LIN {X 0,Y 125.96,Z 856.864,A -85,B 0,C 180,E1 -29175.835,E2 -29175.835} C_VEL
LIN {X 0,Y 122.097,Z 869.522,A -85,B 0,C 180,E1 -29176.604,E2 -29176.604} C_VEL
LIN {X 0,Y 116.788,Z 882.194,A -85,B 0,C 180,E1 -29177.633,E2 -29177.633} C_VEL
LIN {X 0,Y 110.546,Z 893.75,A -85,B 0,C 180,E1 -29179.056,E2 -29179.056} C_VEL
LIN {X 0,Y 103.315,Z 904.432,A -85,B 0,C 180,E1 -29180.801,E2 -29180.801} C_VEL
LIN {X 0,Y 95.494,Z 914.111,A -85,B 0,C 180,E1 -29183.161,E2 -29183.161} C_VEL
LIN {X 0,Y 86.375,Z 923.456,A -85,B 0,C 180,E1 -29186.565,E2 -29186.565} C_VEL
LIN {X 0,Y 77.748,Z 931.029,A -85,B 0,C 180,E1 -29190.898,E2 -29190.898} C_VEL
LIN {X 0,Y 69.801,Z 937.172,A -85,B 0,C 180,E1 -29196.413,E2 -29196.413} C_VEL
LIN {X 0,Y 62.757,Z 942.089,A -85,B 0,C 180,E1 -29203.354,E2 -29203.354} C_VEL
LIN {X 0,Y 56.919,Z 945.911,A -85,B 0,C 180,E1 -29211.938,E2 -29211.938} C_VEL
LIN {X 0,Y 53.931,Z 947.927,A -85,B 0,C 180,E1 -29218.644,E2 -29218.644} C_VEL
LIN {X 0,Y 50.672,Z 950.661,A -85,B 0,C 180,E1 -29233.952,E2 -29233.952} C_VEL
LIN {X 0,Y 50.511,Z 951.445,A -85,B 0,C 180,E1 -29242.056,E2 -29242.056} C_VEL
LIN {X 0,Y 51.125,Z 951.803,A -85,B 0,C 180,E1 -29250.052,E2 -29250.052} C_VEL
LIN {X 0,Y 50.744,Z 950.876,A -85,B 0,C 180,E1 -29264.189,E2 -29264.189} C_VEL
LIN {X 0,Y 52.243,Z 949.486,A -85,B 0,C 180,E1 -29273.856,E2 -29273.856} C_VEL
LIN {X 0,Y 56.006,Z 946.967,A -85,B 0,C 180,E1 -29284.436,E2 -29284.436} C_VEL
LIN {X 0,Y 61.604,Z 943.508,A -85,B 0,C 180,E1 -29293.252,E2 -29293.252} C_VEL
LIN {X 0,Y 68.709,Z 939.048,A -85,B 0,C 180,E1 -29300.154,E2 -29300.154} C_VEL
LIN {X 0,Y 71.326,Z 937.319,A -85,B 0,C 180,E1 -29302.08,E2 -29302.08} C_VEL
LIN {X 0,Y 72.417,Z 935.739,A -85,B 0,C 180,E1 -29304.388,E2 -29304.388} C_VEL
LIN {X 0,Y 64.144,Z 929.643,A -85,B 0,C 180,E1 -29327.342,E2 -29327.342} C_VEL
LIN {X 0,Y 66.621,Z 924.428,A -85,B 0,C 180,E1 -29346.056,E2 -29346.056} C_VEL
LIN {X 0,Y 72.228,Z 920.62,A -85,B 0,C 180,E1 -29356.973,E2 -29356.973} C_VEL
LIN {X 0,Y 79.37,Z 916.695,A -85,B 0,C 180,E1 -29364.251,E2 -29364.251} C_VEL
LIN {X 0,Y 85.958,Z 913.489,A -85,B 0,C 180,E1 -29369.378,E2 -29369.378} C_VEL
LIN {X 0,Y 89.672,Z 911.586,A -85,B 0,C 180,E1 -29371.415,E2 -29371.415} C_VEL
LIN {X 0,Y 88.137,Z 913.443,A -85,B 0,C 180,E1 -29373.098,E2 -29373.098} C_VEL
LIN {X 0,Y 80.195,Z 920.191,A -85,B 0,C 180,E1 -29377.884,E2 -29377.884} C_VEL
LIN {X 0,Y 73.038,Z 925.543,A -85,B 0,C 180,E1 -29383.758,E2 -29383.758} C_VEL
LIN {X 0,Y 68.621,Z 928.473,A -85,B 0,C 180,E1 -29388.214,E2 -29388.214} C_VEL
LIN {X 0,Y 63.119,Z 931.664,A -85,B 0,C 180,E1 -29394.789,E2 -29394.789} C_VEL
LIN {X 0,Y 59.712,Z 933.322,A -85,B 0,C 180,E1 -29399.034,E2 -29399.034} C_VEL
LIN {X 0,Y 53.34,Z 935.711,A -85,B 0,C 180,E1 -29406.365,E2 -29406.365} C_VEL
LIN {X 0,Y 48.796,Z 937.088,A -85,B 0,C 180,E1 -29413.525,E2 -29413.525} C_VEL
LIN {X 0,Y 46.59,Z 937.681,A -85,B 0,C 180,E1 -29420.091,E2 -29420.091} C_VEL
LIN {X 0,Y 46.223,Z 937.775,A -85,B 0,C 180,E1 -29422.482,E2 -29422.482} C_VEL
LIN {X 0,Y 46.353,Z 937.773,A -85,B 0,C 180,E1 -29438.662,E2 -29438.662} C_VEL
LIN {X 0,Y 47.82,Z 937.194,A -85,B 0,C 180,E1 -29447.034,E2 -29447.034} C_VEL
LIN {X 0,Y 52.969,Z 934.956,A -85,B 0,C 180,E1 -29461.993,E2 -29461.993} C_VEL
LIN {X 0,Y 58.863,Z 932.124,A -85,B 0,C 180,E1 -29470.983,E2 -29470.983} C_VEL
LIN {X 0,Y 65.813,Z 928.288,A -85,B 0,C 180,E1 -29478.31,E2 -29478.31} C_VEL
LIN {X 0,Y 74.181,Z 922.798,A -85,B 0,C 180,E1 -29485.018,E2 -29485.018} C_VEL
LIN {X 0,Y 82.984,Z 915.971,A -85,B 0,C 180,E1 -29490.164,E2 -29490.164} C_VEL
LIN {X 0,Y 91.726,Z 907.926,A -85,B 0,C 180,E1 -29494.12,E2 -29494.12} C_VEL
LIN {X 0,Y 99.199,Z 899.686,A -85,B 0,C 180,E1 -29496.996,E2 -29496.996} C_VEL
LIN {X 0,Y 106.833,Z 889.483,A -85,B 0,C 180,E1 -29499.543,E2 -29499.543} C_VEL
LIN {X 0,Y 112.682,Z 880.047,A -85,B 0,C 180,E1 -29501.229,E2 -29501.229} C_VEL
LIN {X 0,Y 117.281,Z 871.144,A -85,B 0,C 180,E1 -29502.419,E2 -29502.419} C_VEL
LIN {X 0,Y 122.094,Z 859.374,A -85,B 0,C 180,E1 -29503.611,E2 -29503.611} C_VEL
LIN {X 0,Y 125.844,Z 846.575,A -85,B 0,C 180,E1 -29504.721,E2 -29504.721} C_VEL
LIN {X 0,Y 127.634,Z 837.303,A -85,B 0,C 180,E1 -29505.399,E2 -29505.399} C_VEL
LIN {X 0,Y 126.554,Z 833.188,A -85,B 0,C 180,E1 -29509.4,E2 -29509.4} C_VEL
LIN {X 0,Y 125.802,Z 830.534,A -85,B 0,C 180,E1 -29513.182,E2 -29513.182} C_VEL
LIN {X 0,Y 125.399,Z 828.562,A -85,B 0,C 180,E1 -29518.394,E2 -29518.394} C_VEL
LIN {X 0,Y 125.412,Z 829.133,A -85,B 0,C 180,E1 -29521.204,E2 -29521.204} C_VEL
LIN {X 0,Y 125.607,Z 830.225,A -85,B 0,C 180,E1 -29523.709,E2 -29523.709} C_VEL
LIN {X 0,Y 126.013,Z 834.743,A -85,B 0,C 180,E1 -29527.511,E2 -29527.511} C_VEL
LIN {X 0,Y 126.597,Z 840.675,A -85,B 0,C 180,E1 -29531.003,E2 -29531.003} C_VEL
LIN {X 0,Y 126.639,Z 841.245,A -85,B 0,C 180,E1 -29531.267,E2 -29531.267} C_VEL
LIN {X 0,Y 124.687,Z 853.794,A -85,B 0,C 180,E1 -29532.524,E2 -29532.524} C_VEL
LIN {X 0,Y 121.012,Z 866.448,A -85,B 0,C 180,E1 -29533.224,E2 -29533.224} C_VEL
LIN {X 0,Y 115.867,Z 878.975,A -85,B 0,C 180,E1 -29534.064,E2 -29534.064} C_VEL
LIN {X 0,Y 109.95,Z 890.23,A -85,B 0,C 180,E1 -29535.191,E2 -29535.191} C_VEL
LIN {X 0,Y 102.648,Z 901.262,A -85,B 0,C 180,E1 -29536.661,E2 -29536.661} C_VEL
LIN {X 0,Y 94.543,Z 911.298,A -85,B 0,C 180,E1 -29538.697,E2 -29538.697} C_VEL
LIN {X 0,Y 85.004,Z 921.052,A -85,B 0,C 180,E1 -29541.64,E2 -29541.64} C_VEL
LIN {X 0,Y 75.838,Z 928.871,A -85,B 0,C 180,E1 -29545.463,E2 -29545.463} C_VEL
LIN {X 0,Y 68.563,Z 934.267,A -85,B 0,C 180,E1 -29549.478,E2 -29549.478} C_VEL
LIN {X 0,Y 60.542,Z 939.563,A -85,B 0,C 180,E1 -29555.731,E2 -29555.731} C_VEL
LIN {X 0,Y 53.518,Z 943.742,A -85,B 0,C 180,E1 -29563.835,E2 -29563.835} C_VEL
LIN {X 0,Y 47.968,Z 946.908,A -85,B 0,C 180,E1 -29574.194,E2 -29574.194} C_VEL
LIN {X 0,Y 43.825,Z 949.638,A -85,B 0,C 180,E1 -29591.358,E2 -29591.358} C_VEL
LIN {X 0,Y 43.425,Z 950.423,A -85,B 0,C 180,E1 -29600.749,E2 -29600.749} C_VEL
LIN {X 0,Y 44.019,Z 950.789,A -85,B 0,C 180,E1 -29610.061,E2 -29610.061} C_VEL
LIN {X 0,Y 43.801,Z 949.941,A -85,B 0,C 180,E1 -29625.697,E2 -29625.697} C_VEL
LIN {X 0,Y 45.805,Z 948.467,A -85,B 0,C 180,E1 -29637.47,E2 -29637.47} C_VEL
LIN {X 0,Y 50.302,Z 945.951,A -85,B 0,C 180,E1 -29649.021,E2 -29649.021} C_VEL
LIN {X 0,Y 56.65,Z 942.495,A -85,B 0,C 180,E1 -29658.171,E2 -29658.171} C_VEL
LIN {X 0,Y 64.087,Z 938.238,A -85,B 0,C 180,E1 -29664.741,E2 -29664.741} C_VEL
LIN {X 0,Y 63.801,Z 937.55,A -85,B 0,C 180,E1 -29666.58,E2 -29666.58} C_VEL
LIN {X 0,Y 57.709,Z 931.539,A -85,B 0,C 180,E1 -29693.005,E2 -29693.005} C_VEL
LIN {X 0,Y 66.173,Z 924.542,A -85,B 0,C 180,E1 -29718.58,E2 -29718.58} C_VEL
LIN {X 0,Y 77.85,Z 919.066,A -85,B 0,C 180,E1 -29729.77,E2 -29729.77} C_VEL
LIN {X 0,Y 79.132,Z 918.523,A -85,B 0,C 180,E1 -29730.709,E2 -29730.709} C_VEL
LIN {X 0,Y 77.189,Z 920.414,A -85,B 0,C 180,E1 -29733.114,E2 -29733.114} C_VEL
LIN {X 0,Y 68.366,Z 926.547,A -85,B 0,C 180,E1 -29739.5,E2 -29739.5} C_VEL
LIN {X 0,Y 63.553,Z 929.477,A -85,B 0,C 180,E1 -29743.988,E2 -29743.988} C_VEL
LIN {X 0,Y 56.806,Z 933.027,A -85,B 0,C 180,E1 -29751.729,E2 -29751.729} C_VEL
LIN {X 0,Y 53.033,Z 934.846,A -85,B 0,C 180,E1 -29757.932,E2 -29757.932} C_VEL
LIN {X 0,Y 47.849,Z 937.141,A -85,B 0,C 180,E1 -29772.86,E2 -29772.86} C_VEL
LIN {X 0,Y 46.223,Z 937.775,A -85,B 0,C 180,E1 -29782.482,E2 -29782.482} C_VEL
LIN {X 0,Y 45.161,Z 938.065,A -85,B 0,C 180,E1 -29789.784,E2 -29789.784} C_VEL
LIN {X 0,Y 43.227,Z 938.129,A -85,B 0,C 180,E1 -29802.443,E2 -29802.443} C_VEL
LIN {X 0,Y 43.031,Z 937.744,A -85,B 0,C 180,E1 -29813.036,E2 -29813.036} C_VEL
LIN {X 0,Y 44.873,Z 936.848,A -85,B 0,C 180,E1 -29821.669,E2 -29821.669} C_VEL
LIN {X 0,Y 45.325,Z 936.617,A -85,B 0,C 180,E1 -29822.768,E2 -29822.768} C_VEL
LIN {X 0,Y 51.399,Z 934.17,A -85,B 0,C 180,E1 -29833.056,E2 -29833.056} C_VEL
LIN {X 0,Y 58.815,Z 930.661,A -85,B 0,C 180,E1 -29840.883,E2 -29840.883} C_VEL
LIN {X 0,Y 68.575,Z 924.982,A -85,B 0,C 180,E1 -29848.511,E2 -29848.511} C_VEL
LIN {X 0,Y 76.72,Z 919.301,A -85,B 0,C 180,E1 -29853.185,E2 -29853.185} C_VEL
LIN {X 0,Y 85.798,Z 911.83,A -85,B 0,C 180,E1 -29857.061,E2 -29857.061} C_VEL
LIN {X 0,Y 93.556,Z 904.17,A -85,B 0,C 180,E1 -29859.793,E2 -29859.793} C_VEL
LIN {X 0,Y 101.396,Z 894.827,A -85,B 0,C 180,E1 -29862.274,E2 -29862.274} C_VEL
LIN {X 0,Y 108.587,Z 884.423,A -85,B 0,C 180,E1 -29864.206,E2 -29864.206} C_VEL
LIN {X 0,Y 114.83,Z 873.288,A -85,B 0,C 180,E1 -29865.58,E2 -29865.58} C_VEL
LIN {X 0,Y 118.787,Z 864.334,A -85,B 0,C 180,E1 -29866.514,E2 -29866.514} C_VEL
LIN {X 0,Y 122.781,Z 852.78,A -85,B 0,C 180,E1 -29867.478,E2 -29867.478} C_VEL
LIN {X 0,Y 125.431,Z 841.744,A -85,B 0,C 180,E1 -29868.317,E2 -29868.317} C_VEL
LIN {X 0,Y 124.898,Z 838.871,A -85,B 0,C 180,E1 -29871.709,E2 -29871.709} C_VEL
LIN {X 0,Y 124.692,Z 837.34,A -85,B 0,C 180,E1 -29873.933,E2 -29873.933} C_VEL
LIN {X 0,Y 124.479,Z 835.709,A -85,B 0,C 180,E1 -29878.382,E2 -29878.382} C_VEL
LIN {X 0,Y 124.49,Z 836.12,A -85,B 0,C 180,E1 -29880.809,E2 -29880.809} C_VEL
LIN {X 0,Y 124.572,Z 837.021,A -85,B 0,C 180,E1 -29882.728,E2 -29882.728} C_VEL
LIN {X 0,Y 124.685,Z 840.698,A -85,B 0,C 180,E1 -29885.864,E2 -29885.864} C_VEL
LIN {X 0,Y 124.757,Z 844.677,A -85,B 0,C 180,E1 -29888.301,E2 -29888.301} C_VEL
LIN {X 0,Y 122.942,Z 854.393,A -85,B 0,C 180,E1 -29889.356,E2 -29889.356} C_VEL
LIN {X 0,Y 119.094,Z 866.746,A -85,B 0,C 180,E1 -29889.963,E2 -29889.963} C_VEL
LIN {X 0,Y 113.682,Z 879.359,A -85,B 0,C 180,E1 -29890.699,E2 -29890.699} C_VEL
LIN {X 0,Y 107.587,Z 890.414,A -85,B 0,C 180,E1 -29891.662,E2 -29891.662} C_VEL
LIN {X 0,Y 100.842,Z 900.253,A -85,B 0,C 180,E1 -29892.794,E2 -29892.794} C_VEL
LIN {X 0,Y 92.514,Z 910.289,A -85,B 0,C 180,E1 -29894.532,E2 -29894.532} C_VEL
LIN {X 0,Y 82.643,Z 920.038,A -85,B 0,C 180,E1 -29897.046,E2 -29897.046} C_VEL
LIN {X 0,Y 73.06,Z 927.857,A -85,B 0,C 180,E1 -29900.415,E2 -29900.415} C_VEL
LIN {X 0,Y 62.369,Z 935.131,A -85,B 0,C 180,E1 -29905.755,E2 -29905.755} C_VEL
LIN {X 0,Y 53.949,Z 940.05,A -85,B 0,C 180,E1 -29912.238,E2 -29912.238} C_VEL
LIN {X 0,Y 46.497,Z 943.872,A -85,B 0,C 180,E1 -29921.002,E2 -29921.002} C_VEL
LIN {X 0,Y 42.359,Z 945.885,A -85,B 0,C 180,E1 -29928.508,E2 -29928.508} C_VEL
LIN {X 0,Y 37.113,Z 948.617,A -85,B 0,C 180,E1 -29947.824,E2 -29947.824} C_VEL
LIN {X 0,Y 36.375,Z 949.401,A -85,B 0,C 180,E1 -29958.935,E2 -29958.935} C_VEL
LIN {X 0,Y 36.907,Z 949.775,A -85,B 0,C 180,E1 -29970.072,E2 -29970.072} C_VEL
LIN {X 0,Y 36.885,Z 949.005,A -85,B 0,C 180,E1 -29987.697,E2 -29987.697} C_VEL
LIN {X 0,Y 39.625,Z 947.451,A -85,B 0,C 180,E1 -30002.223,E2 -30002.223} C_VEL
LIN {X 0,Y 44.987,Z 944.934,A -85,B 0,C 180,E1 -30014.748,E2 -30014.748} C_VEL
LIN {X 0,Y 52.192,Z 941.484,A -85,B 0,C 180,E1 -30023.976,E2 -30023.976} C_VEL
LIN {X 0,Y 55.747,Z 939.698,A -85,B 0,C 180,E1 -30027.013,E2 -30027.013} C_VEL
LIN {X 0,Y 55.22,Z 939.066,A -85,B 0,C 180,E1 -30029.397,E2 -30029.397} C_VEL
LIN {X 0,Y 51.932,Z 933.136,A -85,B 0,C 180,E1 -30060,E2 -30060} C_VEL
LIN {X 0,Y 60.187,Z 928.004,A -85,B 0,C 180,E1 -30080.793,E2 -30080.793} C_VEL
LIN {X 0,Y 67.05,Z 925.068,A -85,B 0,C 180,E1 -30088.144,E2 -30088.144} C_VEL
LIN {X 0,Y 69.724,Z 923.968,A -85,B 0,C 180,E1 -30090.265,E2 -30090.265} C_VEL
LIN {X 0,Y 66.867,Z 925.895,A -85,B 0,C 180,E1 -30092.704,E2 -30092.704} C_VEL
LIN {X 0,Y 58.89,Z 930.481,A -85,B 0,C 180,E1 -30099.062,E2 -30099.062} C_VEL
LIN {X 0,Y 51.472,Z 934.03,A -85,B 0,C 180,E1 -30106.878,E2 -30106.878} C_VEL
LIN {X 0,Y 47.225,Z 935.849,A -85,B 0,C 180,E1 -30113.4,E2 -30113.4} C_VEL
LIN {X 0,Y 41.185,Z 938.144,A -85,B 0,C 180,E1 -30129.977,E2 -30129.977} C_VEL
LIN {X 0,Y 38.804,Z 938.973,A -85,B 0,C 180,E1 -30149.931,E2 -30149.931} C_VEL
LIN {X 0,Y 41.151,Z 938.197,A -85,B 0,C 180,E1 -30169.902,E2 -30169.902} C_VEL
LIN {X 0,Y 45.325,Z 936.617,A -85,B 0,C 180,E1 -30182.768,E2 -30182.768} C_VEL
LIN {X 0,Y 46.784,Z 935.987,A -85,B 0,C 180,E1 -30187.339,E2 -30187.339} C_VEL
LIN {X 0,Y 50.597,Z 933.565,A -85,B 0,C 180,E1 -30202.399,E2 -30202.399} C_VEL
LIN {X 0,Y 53.137,Z 932.34,A -85,B 0,C 180,E1 -30205.49,E2 -30205.49} C_VEL
LIN {X 0,Y 63.26,Z 927.125,A -85,B 0,C 180,E1 -30212.62,E2 -30212.62} C_VEL
LIN {X 0,Y 72.261,Z 921.391,A -85,B 0,C 180,E1 -30217.398,E2 -30217.398} C_VEL
LIN {X 0,Y 81.705,Z 914.171,A -85,B 0,C 180,E1 -30221.006,E2 -30221.006} C_VEL
LIN {X 0,Y 91.366,Z 905.17,A -85,B 0,C 180,E1 -30223.933,E2 -30223.933} C_VEL
LIN {X 0,Y 99.481,Z 895.826,A -85,B 0,C 180,E1 -30226.132,E2 -30226.132} C_VEL
LIN {X 0,Y 106.888,Z 885.422,A -85,B 0,C 180,E1 -30227.834,E2 -30227.834} C_VEL
LIN {X 0,Y 113.284,Z 874.285,A -85,B 0,C 180,E1 -30229.025,E2 -30229.025} C_VEL
LIN {X 0,Y 117.695,Z 864.514,A -85,B 0,C 180,E1 -30229.912,E2 -30229.912} C_VEL
LIN {X 0,Y 121.75,Z 852.71,A -85,B 0,C 180,E1 -30230.804,E2 -30230.804} C_VEL
LIN {X 0,Y 123.369,Z 846.422,A -85,B 0,C 180,E1 -30231.276,E2 -30231.276} C_VEL
LIN {X 0,Y 123.267,Z 844.134,A -85,B 0,C 180,E1 -30234.684,E2 -30234.684} C_VEL
LIN {X 0,Y 123.277,Z 842.806,A -85,B 0,C 180,E1 -30238.366,E2 -30238.366} C_VEL
LIN {X 0,Y 123.316,Z 843.357,A -85,B 0,C 180,E1 -30241.224,E2 -30241.224} C_VEL
LIN {X 0,Y 123.159,Z 846.599,A -85,B 0,C 180,E1 -30244.194,E2 -30244.194} C_VEL
LIN {X 0,Y 123.018,Z 848.51,A -85,B 0,C 180,E1 -30245.424,E2 -30245.424} C_VEL
LIN {X 0,Y 121.014,Z 856.916,A -85,B 0,C 180,E1 -30246.228,E2 -30246.228} C_VEL
LIN {X 0,Y 116.539,Z 869.687,A -85,B 0,C 180,E1 -30246.729,E2 -30246.729} C_VEL
LIN {X 0,Y 111.24,Z 880.928,A -85,B 0,C 180,E1 -30247.283,E2 -30247.283} C_VEL
LIN {X 0,Y 103.804,Z 893.318,A -85,B 0,C 180,E1 -30248.245,E2 -30248.245} C_VEL
LIN {X 0,Y 96.081,Z 903.516,A -85,B 0,C 180,E1 -30249.277,E2 -30249.277} C_VEL
LIN {X 0,Y 87.585,Z 912.759,A -85,B 0,C 180,E1 -30250.777,E2 -30250.777} C_VEL
LIN {X 0,Y 77.489,Z 921.794,A -85,B 0,C 180,E1 -30253.014,E2 -30253.014} C_VEL
LIN {X 0,Y 67.607,Z 929.121,A -85,B 0,C 180,E1 -30256.091,E2 -30256.091} C_VEL
LIN {X 0,Y 56.51,Z 935.87,A -85,B 0,C 180,E1 -30261.272,E2 -30261.272} C_VEL
LIN {X 0,Y 47.59,Z 940.404,A -85,B 0,C 180,E1 -30267.746,E2 -30267.746} C_VEL
LIN {X 0,Y 39.628,Z 943.894,A -85,B 0,C 180,E1 -30277.17,E2 -30277.17} C_VEL
LIN {X 0,Y 33.324,Z 946.421,A -85,B 0,C 180,E1 -30290.857,E2 -30290.857} C_VEL
LIN {X 0,Y 29.377,Z 948.38,A -85,B 0,C 180,E1 -30316.253,E2 -30316.253} C_VEL
LIN {X 0,Y 29.792,Z 948.76,A -85,B 0,C 180,E1 -30330.09,E2 -30330.09} C_VEL
LIN {X 0,Y 30.03,Z 948.053,A -85,B 0,C 180,E1 -30350.589,E2 -30350.589} C_VEL
LIN {X 0,Y 33.805,Z 946.433,A -85,B 0,C 180,E1 -30368.685,E2 -30368.685} C_VEL
LIN {X 0,Y 40.244,Z 943.917,A -85,B 0,C 180,E1 -30381.902,E2 -30381.902} C_VEL
LIN {X 0,Y 46.669,Z 941.24,A -85,B 0,C 180,E1 -30389.291,E2 -30389.291} C_VEL
LIN {X 0,Y 46.791,Z 940.266,A -85,B 0,C 180,E1 -30393.218,E2 -30393.218} C_VEL
LIN {X 0,Y 45.224,Z 935.985,A -85,B 0,C 180,E1 -30420,E2 -30420} C_VEL
LIN {X 0,Y 53.824,Z 931.224,A -85,B 0,C 180,E1 -30443.062,E2 -30443.062} C_VEL
LIN {X 0,Y 58.442,Z 929.439,A -85,B 0,C 180,E1 -30448.753,E2 -30448.753} C_VEL
LIN {X 0,Y 57.514,Z 930.111,A -85,B 0,C 180,E1 -30451.115,E2 -30451.115} C_VEL
LIN {X 0,Y 49.199,Z 933.99,A -85,B 0,C 180,E1 -30458.135,E2 -30458.135} C_VEL
LIN {X 0,Y 41.793,Z 936.853,A -85,B 0,C 180,E1 -30467.645,E2 -30467.645} C_VEL
LIN {X 0,Y 34.666,Z 939.147,A -85,B 0,C 180,E1 -30485.997,E2 -30485.997} C_VEL
LIN {X 0,Y 31.776,Z 939.976,A -85,B 0,C 180,E1 -30509.916,E2 -30509.916} C_VEL
LIN {X 0,Y 34.626,Z 939.199,A -85,B 0,C 180,E1 -30533.864,E2 -30533.864} C_VEL
LIN {X 0,Y 41.717,Z 936.96,A -85,B 0,C 180,E1 -30552.277,E2 -30552.277} C_VEL
LIN {X 0,Y 49.125,Z 934.128,A -85,B 0,C 180,E1 -30561.799,E2 -30561.799} C_VEL
LIN {X 0,Y 53.137,Z 932.34,A -85,B 0,C 180,E1 -30565.49,E2 -30565.49} C_VEL
LIN {X 0,Y 57.264,Z 930.32,A -85,B 0,C 180,E1 -30569.316,E2 -30569.316} C_VEL
LIN {X 0,Y 60.88,Z 928.292,A -85,B 0,C 180,E1 -30573.45,E2 -30573.45} C_VEL
LIN {X 0,Y 69.445,Z 922.785,A -85,B 0,C 180,E1 -30581.842,E2 -30581.842} C_VEL
LIN {X 0,Y 73.748,Z 919.722,A -85,B 0,C 180,E1 -30583.992,E2 -30583.992} C_VEL
LIN {X 0,Y 83.011,Z 912.382,A -85,B 0,C 180,E1 -30586.655,E2 -30586.655} C_VEL
LIN {X 0,Y 91.337,Z 904.432,A -85,B 0,C 180,E1 -30588.66,E2 -30588.66} C_VEL
LIN {X 0,Y 99.723,Z 894.724,A -85,B 0,C 180,E1 -30590.442,E2 -30590.442} C_VEL
LIN {X 0,Y 107.119,Z 884.103,A -85,B 0,C 180,E1 -30591.815,E2 -30591.815} C_VEL
LIN {X 0,Y 112.719,Z 874.135,A -85,B 0,C 180,E1 -30592.69,E2 -30592.69} C_VEL
LIN {X 0,Y 117.701,Z 862.861,A -85,B 0,C 180,E1 -30593.469,E2 -30593.469} C_VEL
LIN {X 0,Y 121.424,Z 851.544,A -85,B 0,C 180,E1 -30594.289,E2 -30594.289} C_VEL
LIN {X 0,Y 121.536,Z 850.559,A -85,B 0,C 180,E1 -30596.228,E2 -30596.228} C_VEL
LIN {X 0,Y 121.683,Z 849.854,A -85,B 0,C 180,E1 -30598.345,E2 -30598.345} C_VEL
LIN {X 0,Y 121.708,Z 850.206,A -85,B 0,C 180,E1 -30600.517,E2 -30600.517} C_VEL
LIN {X 0,Y 121.391,Z 852.398,A -85,B 0,C 180,E1 -30602.458,E2 -30602.458} C_VEL
LIN {X 0,Y 120.013,Z 857.403,A -85,B 0,C 180,E1 -30602.895,E2 -30602.895} C_VEL
LIN {X 0,Y 115.482,Z 869.689,A -85,B 0,C 180,E1 -30603.273,E2 -30603.273} C_VEL
LIN {X 0,Y 109.561,Z 881.749,A -85,B 0,C 180,E1 -30603.701,E2 -30603.701} C_VEL
LIN {X 0,Y 103.024,Z 892.308,A -85,B 0,C 180,E1 -30604.328,E2 -30604.328} C_VEL
LIN {X 0,Y 95.194,Z 902.505,A -85,B 0,C 180,E1 -30605.05,E2 -30605.05} C_VEL
LIN {X 0,Y 86.539,Z 911.748,A -85,B 0,C 180,E1 -30606.151,E2 -30606.151} C_VEL
LIN {X 0,Y 76.203,Z 920.781,A -85,B 0,C 180,E1 -30607.793,E2 -30607.793} C_VEL
LIN {X 0,Y 65.988,Z 928.107,A -85,B 0,C 180,E1 -30610.139,E2 -30610.139} C_VEL
LIN {X 0,Y 54.32,Z 934.848,A -85,B 0,C 180,E1 -30614.203,E2 -30614.203} C_VEL
LIN {X 0,Y 44.712,Z 939.386,A -85,B 0,C 180,E1 -30619.611,E2 -30619.611} C_VEL
LIN {X 0,Y 35.768,Z 942.876,A -85,B 0,C 180,E1 -30628.015,E2 -30628.015} C_VEL
LIN {X 0,Y 28.139,Z 945.401,A -85,B 0,C 180,E1 -30641.619,E2 -30641.619} C_VEL
LIN {X 0,Y 22.485,Z 947.358,A -85,B 0,C 180,E1 -30671.912,E2 -30671.912} C_VEL
LIN {X 0,Y 22.654,Z 947.741,A -85,B 0,C 180,E1 -30690.118,E2 -30690.118} C_VEL
LIN {X 0,Y 24.797,Z 946.577,A -85,B 0,C 180,E1 -30724.658,E2 -30724.658} C_VEL
LIN {X 0,Y 33.525,Z 943.86,A -85,B 0,C 180,E1 -30747.127,E2 -30747.127} C_VEL
LIN {X 0,Y 39.19,Z 941.859,A -85,B 0,C 180,E1 -30753.868,E2 -30753.868} C_VEL
LIN {X 0,Y 37.784,Z 939.811,A -85,B 0,C 180,E1 -30769.281,E2 -30769.281} C_VEL
LIN {X 0,Y 47.574,Z 933.936,A -85,B 0,C 180,E1 -30806.308,E2 -30806.308} C_VEL
LIN {X 0,Y 48.12,Z 933.801,A -85,B 0,C 180,E1 -30808.691,E2 -30808.691} C_VEL
LIN {X 0,Y 42.318,Z 936.037,A -85,B 0,C 180,E1 -30813.755,E2 -30813.755} C_VEL
LIN {X 0,Y 36.904,Z 937.856,A -85,B 0,C 180,E1 -30820.273,E2 -30820.273} C_VEL
LIN {X 0,Y 28.39,Z 940.15,A -85,B 0,C 180,E1 -30840.217,E2 -30840.217} C_VEL
LIN {X 0,Y 24.748,Z 940.978,A -85,B 0,C 180,E1 -30869.892,E2 -30869.892} C_VEL
LIN {X 0,Y 28.341,Z 940.201,A -85,B 0,C 180,E1 -30899.622,E2 -30899.622} C_VEL
LIN {X 0,Y 36.821,Z 937.962,A -85,B 0,C 180,E1 -30919.654,E2 -30919.654} C_VEL
LIN {X 0,Y 45.118,Z 935.13,A -85,B 0,C 180,E1 -30928.83,E2 -30928.83} C_VEL
LIN {X 0,Y 54.13,Z 931.292,A -85,B 0,C 180,E1 -30935.219,E2 -30935.219} C_VEL
LIN {X 0,Y 64.451,Z 925.801,A -85,B 0,C 180,E1 -30940.565,E2 -30940.565} C_VEL
LIN {X 0,Y 73.748,Z 919.722,A -85,B 0,C 180,E1 -30943.992,E2 -30943.992} C_VEL
LIN {X 0,Y 78.012,Z 916.488,A -85,B 0,C 180,E1 -30945.846,E2 -30945.846} C_VEL
LIN {X 0,Y 84.397,Z 911.045,A -85,B 0,C 180,E1 -30949.591,E2 -30949.591} C_VEL
LIN {X 0,Y 90.639,Z 905.012,A -85,B 0,C 180,E1 -30952.751,E2 -30952.751} C_VEL
LIN {X 0,Y 94.511,Z 900.824,A -85,B 0,C 180,E1 -30953.8,E2 -30953.8} C_VEL
LIN {X 0,Y 102.243,Z 891.174,A -85,B 0,C 180,E1 -30954.99,E2 -30954.99} C_VEL
LIN {X 0,Y 108.308,Z 881.913,A -85,B 0,C 180,E1 -30955.764,E2 -30955.764} C_VEL
LIN {X 0,Y 114.08,Z 870.993,A -85,B 0,C 180,E1 -30956.539,E2 -30956.539} C_VEL
LIN {X 0,Y 118.88,Z 859.053,A -85,B 0,C 180,E1 -30957.149,E2 -30957.149} C_VEL
LIN {X 0,Y 119.551,Z 857.065,A -85,B 0,C 180,E1 -30957.324,E2 -30957.324} C_VEL
LIN {X 0,Y 119.425,Z 857.713,A -85,B 0,C 180,E1 -30959.52,E2 -30959.52} C_VEL
LIN {X 0,Y 114.184,Z 871.21,A -85,B 0,C 180,E1 -30959.794,E2 -30959.794} C_VEL
LIN {X 0,Y 108.605,Z 882.057,A -85,B 0,C 180,E1 -30960.011,E2 -30960.011} C_VEL
LIN {X 0,Y 101.855,Z 892.549,A -85,B 0,C 180,E1 -30960.418,E2 -30960.418} C_VEL
LIN {X 0,Y 93.079,Z 903.466,A -85,B 0,C 180,E1 -30960.877,E2 -30960.877} C_VEL
LIN {X 0,Y 84.315,Z 912.385,A -85,B 0,C 180,E1 -30961.579,E2 -30961.579} C_VEL
LIN {X 0,Y 73.82,Z 921.102,A -85,B 0,C 180,E1 -30962.636,E2 -30962.636} C_VEL
LIN {X 0,Y 63.375,Z 928.136,A -85,B 0,C 180,E1 -30964.251,E2 -30964.251} C_VEL
LIN {X 0,Y 53.019,Z 933.827,A -85,B 0,C 180,E1 -30966.675,E2 -30966.675} C_VEL
LIN {X 0,Y 42.845,Z 938.366,A -85,B 0,C 180,E1 -30970.565,E2 -30970.565} C_VEL
LIN {X 0,Y 33.01,Z 941.852,A -85,B 0,C 180,E1 -30976.943,E2 -30976.943} C_VEL
LIN {X 0,Y 23.978,Z 944.377,A -85,B 0,C 180,E1 -30988.684,E2 -30988.684} C_VEL
LIN {X 0,Y 15.853,Z 946.34,A -85,B 0,C 180,E1 -31023.873,E2 -31023.873} C_VEL
LIN {X 0,Y 15.518,Z 946.723,A -85,B 0,C 180,E1 -31050.172,E2 -31050.172} C_VEL
LIN {X 0,Y 19.369,Z 945.561,A -85,B 0,C 180,E1 -31096.724,E2 -31096.724} C_VEL
LIN {X 0,Y 30.255,Z 942.842,A -85,B 0,C 180,E1 -31118.536,E2 -31118.536} C_VEL
LIN {X 0,Y 30.957,Z 941.762,A -85,B 0,C 180,E1 -31126.878,E2 -31126.878} C_VEL
LIN {X 0,Y 37.711,Z 937.427,A -85,B 0,C 180,E1 -31164.008,E2 -31164.008} C_VEL
LIN {X 0,Y 36.679,Z 937.738,A -85,B 0,C 180,E1 -31166.961,E2 -31166.961} C_VEL
LIN {X 0,Y 27.277,Z 940.204,A -85,B 0,C 180,E1 -31179.229,E2 -31179.229} C_VEL
LIN {X 0,Y 22.562,Z 941.153,A -85,B 0,C 180,E1 -31191.316,E2 -31191.316} C_VEL
LIN {X 0,Y 17.721,Z 941.981,A -85,B 0,C 180,E1 -31229.849,E2 -31229.849} C_VEL
LIN {X 0,Y 22.502,Z 941.204,A -85,B 0,C 180,E1 -31268.503,E2 -31268.503} C_VEL
LIN {X 0,Y 32.713,Z 938.964,A -85,B 0,C 180,E1 -31289.079,E2 -31289.079} C_VEL
LIN {X 0,Y 41.914,Z 936.131,A -85,B 0,C 180,E1 -31297.079,E2 -31297.079} C_VEL
LIN {X 0,Y 51.581,Z 932.294,A -85,B 0,C 180,E1 -31302.326,E2 -31302.326} C_VEL
LIN {X 0,Y 62.465,Z 926.802,A -85,B 0,C 180,E1 -31306.655,E2 -31306.655} C_VEL
LIN {X 0,Y 73.181,Z 919.974,A -85,B 0,C 180,E1 -31309.629,E2 -31309.629} C_VEL
LIN {X 0,Y 83.384,Z 911.927,A -85,B 0,C 180,E1 -31311.778,E2 -31311.778} C_VEL
LIN {X 0,Y 91.93,Z 903.685,A -85,B 0,C 180,E1 -31313.346,E2 -31313.346} C_VEL
LIN {X 0,Y 94.511,Z 900.824,A -85,B 0,C 180,E1 -31313.8,E2 -31313.8} C_VEL
LIN {X 0,Y 93.564,Z 901.914,A -85,B 0,C 180,E1 -31314.335,E2 -31314.335} C_VEL
LIN {X 0,Y 88.039,Z 907.77,A -85,B 0,C 180,E1 -31315.002,E2 -31315.002} C_VEL
LIN {X 0,Y 78.788,Z 916.053,A -85,B 0,C 180,E1 -31315.222,E2 -31315.222} C_VEL
LIN {X 0,Y 73.915,Z 919.79,A -85,B 0,C 180,E1 -31315.084,E2 -31315.084} C_VEL
LIN {X 0,Y 68.872,Z 923.242,A -85,B 0,C 180,E1 -31314.593,E2 -31314.593} C_VEL
LIN {X 0,Y 58.982,Z 928.987,A -85,B 0,C 180,E1 -31312.492,E2 -31312.492} C_VEL
LIN {X 0,Y 46.51,Z 934.667,A -85,B 0,C 180,E1 -31308.849,E2 -31308.849} C_VEL
LIN {X 0,Y 36.34,Z 938.177,A -85,B 0,C 180,E1 -31304.936,E2 -31304.936} C_VEL
LIN {X 0,Y 29.719,Z 939.966,A -85,B 0,C 180,E1 -31300.785,E2 -31300.785} C_VEL
LIN {X 0,Y 17.556,Z 942.206,A -85,B 0,C 180,E1 -31282.935,E2 -31282.935} C_VEL
LIN {X 0,Y 10.693,Z 942.984,A -85,B 0,C 180,E1 -31229.75,E2 -31229.75} C_VEL
LIN {X 0,Y 17.631,Z 942.156,A -85,B 0,C 180,E1 -31176.889,E2 -31176.889} C_VEL
LIN {X 0,Y 25.49,Z 940.814,A -85,B 0,C 180,E1 -31163.348,E2 -31163.348} C_VEL
LIN {X 0,Y 27.347,Z 940.503,A -85,B 0,C 180,E1 -31158.252,E2 -31158.252} C_VEL
LIN {X 0,Y 24.026,Z 942.512,A -85,B 0,C 180,E1 -31134.013,E2 -31134.013} C_VEL
LIN {X 0,Y 23.017,Z 943.12,A -85,B 0,C 180,E1 -31127.979,E2 -31127.979} C_VEL
LIN {X 0,Y 11.275,Z 945.164,A -85,B 0,C 180,E1 -31101.442,E2 -31101.442} C_VEL
LIN {X 0,Y 8.369,Z 945.703,A -85,B 0,C 180,E1 -31050.319,E2 -31050.319} C_VEL
LIN {X 0,Y 10.019,Z 945.301,A -85,B 0,C 180,E1 -31004.543,E2 -31004.543} C_VEL
LIN {X 0,Y 21.48,Z 943.356,A -85,B 0,C 180,E1 -30971.676,E2 -30971.676} C_VEL
LIN {X 0,Y 31.672,Z 940.83,A -85,B 0,C 180,E1 -30964.44,E2 -30964.44} C_VEL
LIN {X 0,Y 42.124,Z 937.348,A -85,B 0,C 180,E1 -30960.964,E2 -30960.964} C_VEL
LIN {X 0,Y 52.669,Z 932.81,A -85,B 0,C 180,E1 -30958.942,E2 -30958.942} C_VEL
LIN {X 0,Y 64.832,Z 926.19,A -85,B 0,C 180,E1 -30957.71,E2 -30957.71} C_VEL
LIN {X 0,Y 75.6,Z 918.755,A -85,B 0,C 180,E1 -30957.042,E2 -30957.042} C_VEL
LIN {X 0,Y 77.365,Z 917.372,A -85,B 0,C 180,E1 -30956.957,E2 -30956.957} C_VEL
LIN {X 0,Y 77.452,Z 917.172,A -85,B 0,C 180,E1 -30955.922,E2 -30955.922} C_VEL
LIN {X 0,Y 68.872,Z 923.242,A -85,B 0,C 180,E1 -30954.593,E2 -30954.593} C_VEL
LIN {X 0,Y 67.964,Z 924.927,A -85,B 0,C 180,E1 -30954.461,E2 -30954.461} C_VEL
LIN {X 0,Y 67.964,Z 952.182,A -85,B 0,C 180,E1 -30954.461,E2 -30954.461} C_VEL
LIN {X 0,Y 23.687,Z 952.182,A -85,B 0,C 180,E1 -30946.529,E2 -30946.529} C_VEL
LIN {X 0,Y 21.736,Z 950.182,A -85,B 0,C 180,E1 -30945.42,E2 -30945.42} C_VEL
LIN {X 0,Y 21.736,Z 944.261,A -85,B 0,C 180,E1 -30945.42,E2 -30945.42} C_VEL
LIN {X 0,Y 21.276,Z 942.281,A -85,B 0,C 180,E1 -30951.379,E2 -30951.379} C_VEL
LIN {X 0,Y 21.224,Z 942.333,A -85,B 0,C 180,E1 -30952.358,E2 -30952.358} C_VEL
LIN {X 0,Y 6.517,Z 944.341,A -85,B 0,C 180,E1 -30959.997,E2 -30959.997} C_VEL
LIN {X 0,Y 1.224,Z 944.684,A -85,B 0,C 180,E1 -31052.182,E2 -31052.182} C_VEL
LIN {X 0,Y 8.22,Z 944.202,A -85,B 0,C 180,E1 -31140.003,E2 -31140.003} C_VEL
LIN {X 0,Y 14.136,Z 943.525,A -85,B 0,C 180,E1 -31144.017,E2 -31144.017} C_VEL
LIN {X 0,Y 17.773,Z 942.902,A -85,B 0,C 180,E1 -31147.348,E2 -31147.348} C_VEL
LIN {X 0,Y 14.543,Z 943.159,A -85,B 0,C 180,E1 -31154.152,E2 -31154.152} C_VEL
LIN {X 0,Y 3.665,Z 943.986,A -85,B 0,C 180,E1 -31229.271,E2 -31229.271} C_VEL
LIN {X 0,Y 14.452,Z 943.208,A -85,B 0,C 180,E1 -31305.768,E2 -31305.768} C_VEL
LIN {X 0,Y 21.276,Z 942.281,A -85,B 0,C 180,E1 -31311.379,E2 -31311.379} C_VEL
LIN {X 0,Y 21.276,Z 942.281,A -85,B 0,C 180,E1 -31311.379,E2 -31311.379}

QRS_NEXT_CUT()

QRS_NEXT()
QRS_HOME()

END
